{attribute addProperty BoxType "EP6224-0002-0016"}
{attribute addProperty Id "Module_1_DeviceState_Inputs_DeviceModule_1_DeviceState_Inputs_Device_50DD3C951620Module_2_DeviceState_InputsModule_2_DeviceState_Inputs_D860B2E33240Module_7_Digital_InputsModule_7_Digital_Inputs_AB7F33C83240WcStateAT %I*WcState_98A4DF7520.250InfoDataAT %I*InfoData_275E3363128160"}
{attribute addProperty CRC "3265840221"}
{attribute addProperty SizeInBites "210"}
{attribute addProperty SizeInBytes "26.25"}
TYPE EP6224_69FFDAE7 :
STRUCT
	{attribute addProperty Name "Module_1_DeviceState_Inputs_Device"}
	Module_1_DeviceState_Inputs_Device : Module_1_DeviceState_Inputs_Device_50DD3C95;
	{attribute addProperty Name "Module_2_DeviceState_Inputs"}
	Module_2_DeviceState_Inputs : Module_2_DeviceState_Inputs_D860B2E3;
	{attribute addProperty Name "Module_7_Digital_Inputs"}
	Module_7_Digital_Inputs : Module_7_Digital_Inputs_AB7F33C8;
	{attribute addProperty Name "WcState"}
	WcState : WcState_98A4DF75;
	{attribute addProperty Name "InfoData"}
	InfoData : InfoData_275E3363;
END_STRUCT
END_TYPE

(* stored: Version 1.2.0.0, ProductVersion 3.1.4024.9
   DUT EP6224_69FFDAE7: Id {239dfda4-93ad-4b95-819c-7a69f57793b4} *)
